FUNCTION_BLOCK "FB_Dispatch_Point_T"
TITLE = %version: 5.09 % %Commit:  c3808b61 % CN: 50
{ S7_Optimized_Access := 'FALSE' }
FAMILY : Tubtrax
VERSION : 0.0
//Function:
//Dispatch point is used to assign carriers up to 15 different destinations using
//balance load criteria.
//
BEGIN
NETWORK
TITLE = AA: Some network title
      NOP 0;

// Copy section event DB number
      OPN "DB_Event_Section";

      L DBNO;
      T #t_DB_Event_Section;

NETWORK
TITLE = BB: Some network title out of order
      NOP 0;

// Copy section event DB number
      OPN "DB_Event_Section";

      L DBNO;
      T #t_DB_Event_Section;

NETWORK
TITLE = AB: Some network title taking the blame
      NOP 0;

// Copy section event DB number
      OPN "DB_Event_Section";

      L DBNO;
      T #t_DB_Event_Section;

NETWORK
TITLE = AC: Good
      NOP 0;

// Copy section event DB number
      OPN "DB_Event_Section";

      L DBNO;
      T #t_DB_Event_Section;

END_FUNCTION_BLOCK
